(* Schneider Machine Expert - Basic project Proiect_final, file version 2.6.0.0 *)
(* ProjectInformations: Name=New project *)

HARDWARE
  Cpu 0: TM221CE16R
  ModuleExtensionObject 0: TM3AM6/G
  EthernetConfiguration: NetworkName=M221, IpAllocationMode=FixedAddress, IpAddress=0.0.0.0, SubnetMask=0.0.0.0
  SerialLineConfiguration: Baud=Baud19200, Parity=ParityEven, DataBits=DataBits8, StopBits=StopBits1, PhysicalMedium=PhysicalMediumRs485, TransmissionMode=TransmissionModeModbusRtu, SlaveId=1, Addressing=SlaveAddressing
  MastTask: UsePeriodScanMode=false, PeriodScan=100
  FastTask: Period=255
  CpuBehavior: StartingMode=StartAsPreviousState, AutoSaveRamOnEeprom=true, WatchdogPeriod=250

SYMBOLS  (address, symbol, comment, settings)
  %M0         "Plata_card"
  %M1         "Plata_cash"
  %M2         "Oltenia"
  %M3         "Moldova"
  %M4         "Transilvania"
  %M5         "Dobrogea"
  %M6         "Trece_banconte_de_50"
  %M7         "Trece_bancnote_de_5"
  %M8         "Trece_bancnote_de_10"
  %M9         "Trece_bancnote_de_1"
  %M10        "Plata_a_fost_facuta"
  %M11        "PLATA_CARD_A_FOST_FACUTA"
  %M12        "A_FOST_SELECTAT_CEVA"
  %C0         "Numarator_50_lei"
  %C1         "Numarator_10_lei"
  %C2         "Numarator_5_lei"
  %C3         "Numarator_1_leu"
  %I0.0       "Pornire selectie"
  %I0.1       "Plata_card"
  %I0.2       "Plata_cash"
  %I0.3       "Selecteaza_Oltenia"
  %I0.4       "Selecteaza_Moldova"
  %I0.5       "Selecteaza_Transilvania"
  %I0.6       "Selecteaza_Dobrogea"
  %I0.8       "SENZOR_A_FOST_LIVRAT_TICHETUL"
  %Q0.0       "S-a eliberat tichetul"
  %IW1.0      [Type=Type_4_20mA, Scope=Scope_Customized, Minimum=4000, Maximum=20000]
  %IW1.1      [Type=Type_4_20mA, Scope=Scope_Customized, Minimum=4000, Maximum=20000]

POU New POU
  (* SectionNumber=1 *)

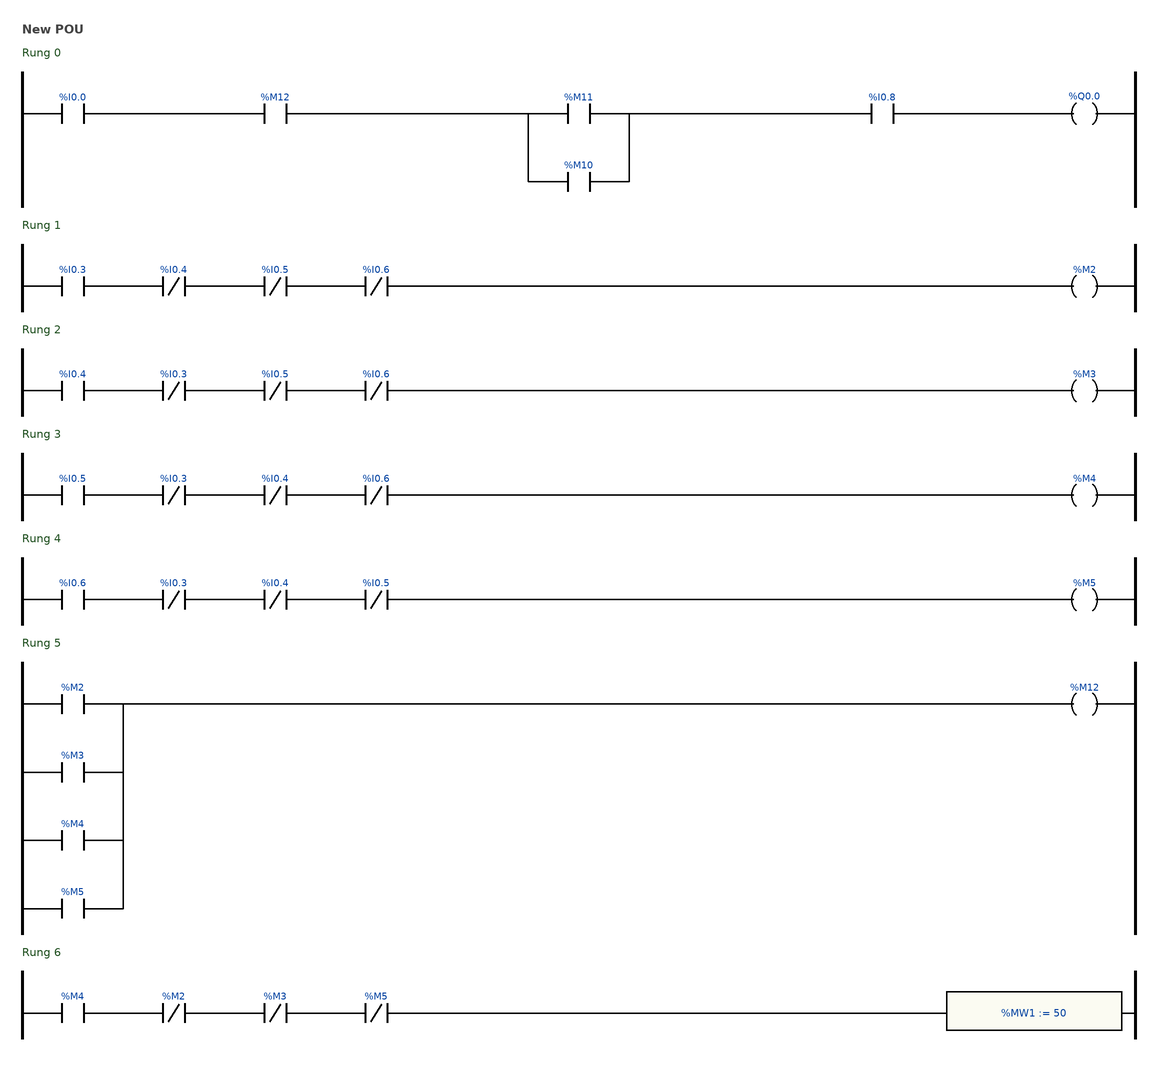

// Rung 0
  LD %I0.0
  AND %M12
  AND( %M11
  OR %M10
  )
  AND %I0.8
  ST %Q0.0
  // as ST:
  //   %Q0.0 := %I0.0 AND %M12 AND (%M11 OR %M10) AND %I0.8;

// Rung 1
  LD %I0.3
  ANDN %I0.4
  ANDN %I0.5
  ANDN %I0.6
  ST %M2
  // as ST:
  //   %M2 := %I0.3 AND NOT %I0.4 AND NOT %I0.5 AND NOT %I0.6;

// Rung 2
  LD %I0.4
  ANDN %I0.3
  ANDN %I0.5
  ANDN %I0.6
  ST %M3
  // as ST:
  //   %M3 := %I0.4 AND NOT %I0.3 AND NOT %I0.5 AND NOT %I0.6;

// Rung 3
  LD %I0.5
  ANDN %I0.3
  ANDN %I0.4
  ANDN %I0.6
  ST %M4
  // as ST:
  //   %M4 := %I0.5 AND NOT %I0.3 AND NOT %I0.4 AND NOT %I0.6;

// Rung 4
  LD %I0.6
  ANDN %I0.3
  ANDN %I0.4
  ANDN %I0.5
  ST %M5
  // as ST:
  //   %M5 := %I0.6 AND NOT %I0.3 AND NOT %I0.4 AND NOT %I0.5;

// Rung 5
  LD %M2
  OR %M3
  OR %M4
  OR %M5
  ST %M12
  // as ST:
  //   %M12 := %M2 OR %M3 OR %M4 OR %M5;

// Rung 6
  LD %M4
  ANDN %M2
  ANDN %M3
  ANDN %M5
  [ %MW1 := 50 ]
  // as ST:
  //   IF %M4 AND NOT %M2 AND NOT %M3 AND NOT %M5 THEN %MW1 := 50; END_IF;

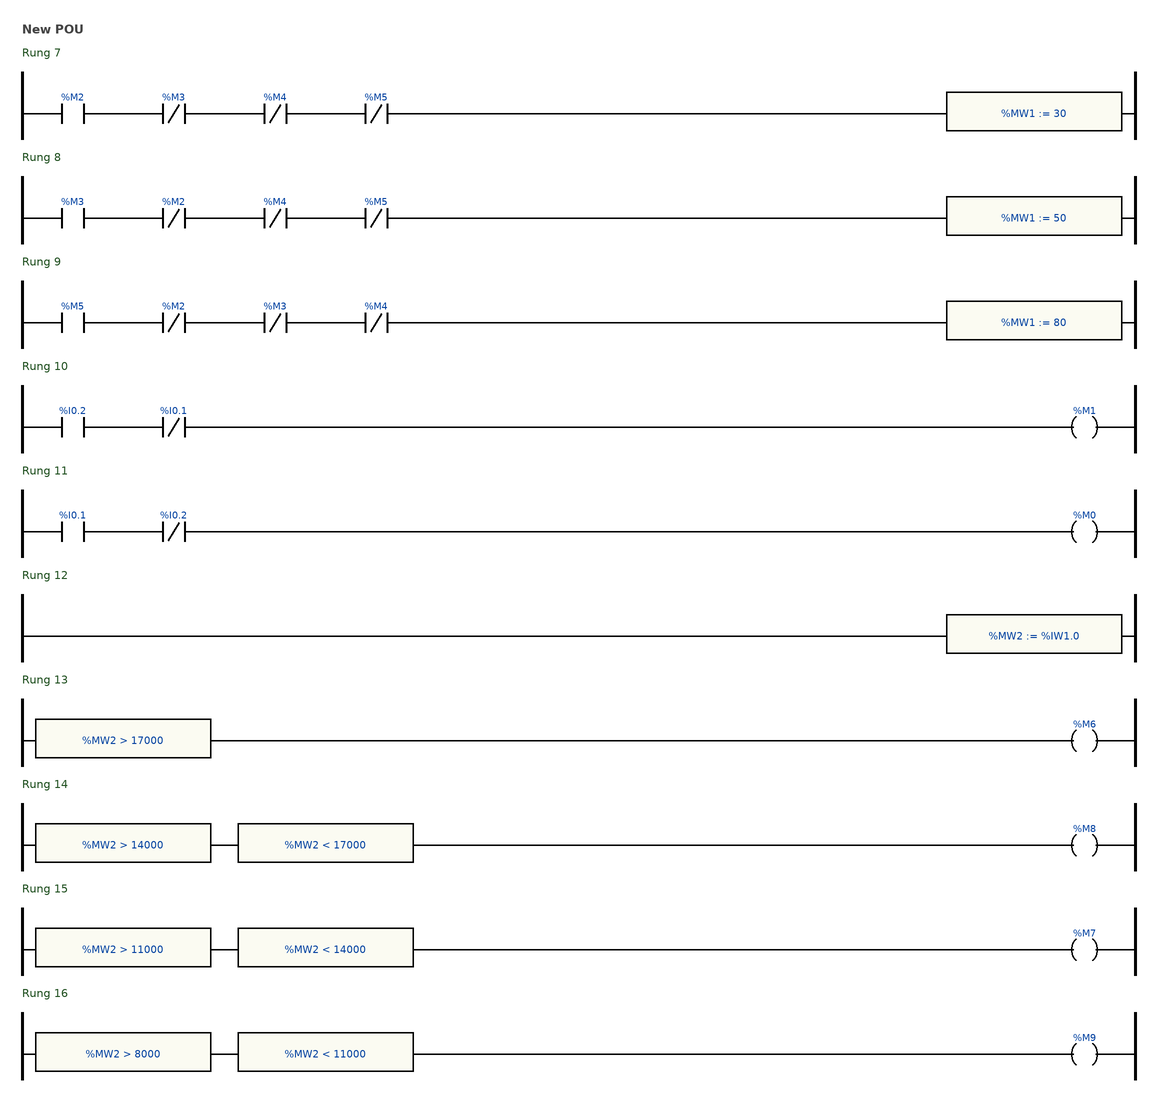

// Rung 7
  LD %M2
  ANDN %M3
  ANDN %M4
  ANDN %M5
  [ %MW1 := 30 ]
  // as ST:
  //   IF %M2 AND NOT %M3 AND NOT %M4 AND NOT %M5 THEN %MW1 := 30; END_IF;

// Rung 8
  LD %M3
  ANDN %M2
  ANDN %M4
  ANDN %M5
  [ %MW1 := 50 ]
  // as ST:
  //   IF %M3 AND NOT %M2 AND NOT %M4 AND NOT %M5 THEN %MW1 := 50; END_IF;

// Rung 9
  LD %M5
  ANDN %M2
  ANDN %M3
  ANDN %M4
  [ %MW1 := 80 ]
  // as ST:
  //   IF %M5 AND NOT %M2 AND NOT %M3 AND NOT %M4 THEN %MW1 := 80; END_IF;

// Rung 10
  LD %I0.2
  ANDN %I0.1
  ST %M1
  // as ST:
  //   %M1 := %I0.2 AND NOT %I0.1;

// Rung 11
  LD %I0.1
  ANDN %I0.2
  ST %M0
  // as ST:
  //   %M0 := %I0.1 AND NOT %I0.2;

// Rung 12
  LD 1
  [ %MW2 := %IW1.0 ]
  // as ST:
  //   %MW2 := %IW1.0;

// Rung 13
  LD [ %MW2 > 17000 ]
  ST %M6
  // as ST:
  //   %M6 := %MW2 > 17000;

// Rung 14
  LD [ %MW2 > 14000 ]
  AND [ %MW2 < 17000 ]
  ST %M8
  // as ST:
  //   %M8 := %MW2 > 14000 AND %MW2 < 17000;

// Rung 15
  LD [ %MW2 > 11000 ]
  AND [ %MW2 < 14000 ]
  ST %M7
  // as ST:
  //   %M7 := %MW2 > 11000 AND %MW2 < 14000;

// Rung 16
  LD [ %MW2 > 8000 ]
  AND [ %MW2 < 11000 ]
  ST %M9
  // as ST:
  //   %M9 := %MW2 > 8000 AND %MW2 < 11000;

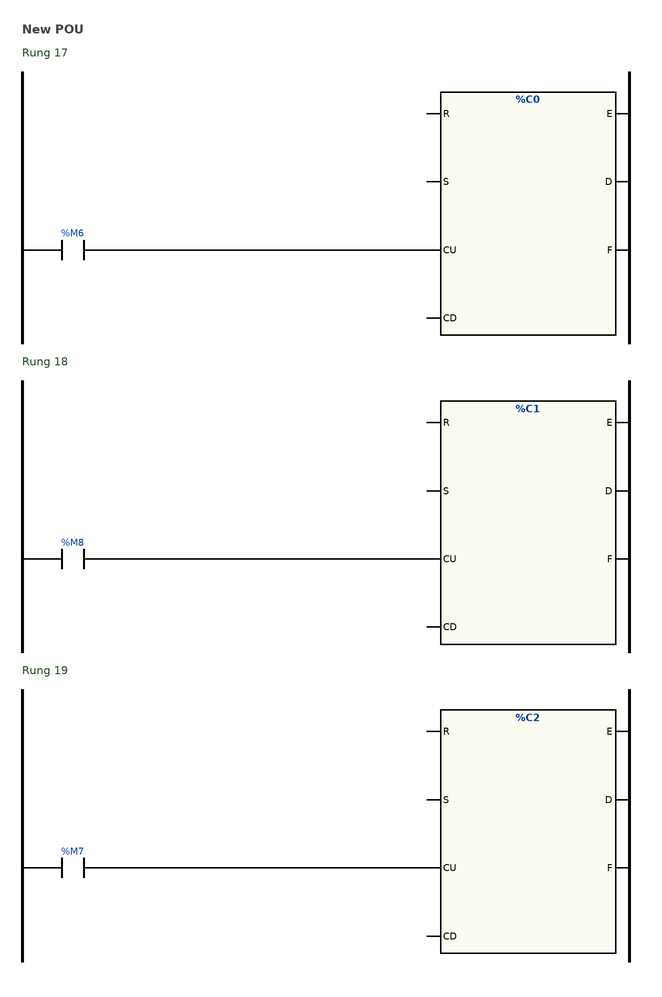

// Rung 17
  BLK %C0
  LD %M6
  CU
  END_BLK
  // as ST:
  //   %C0(CU := %M6);

// Rung 18
  BLK %C1
  LD %M8
  CU
  END_BLK
  // as ST:
  //   %C1(CU := %M8);

// Rung 19
  BLK %C2
  LD %M7
  CU
  END_BLK
  // as ST:
  //   %C2(CU := %M7);

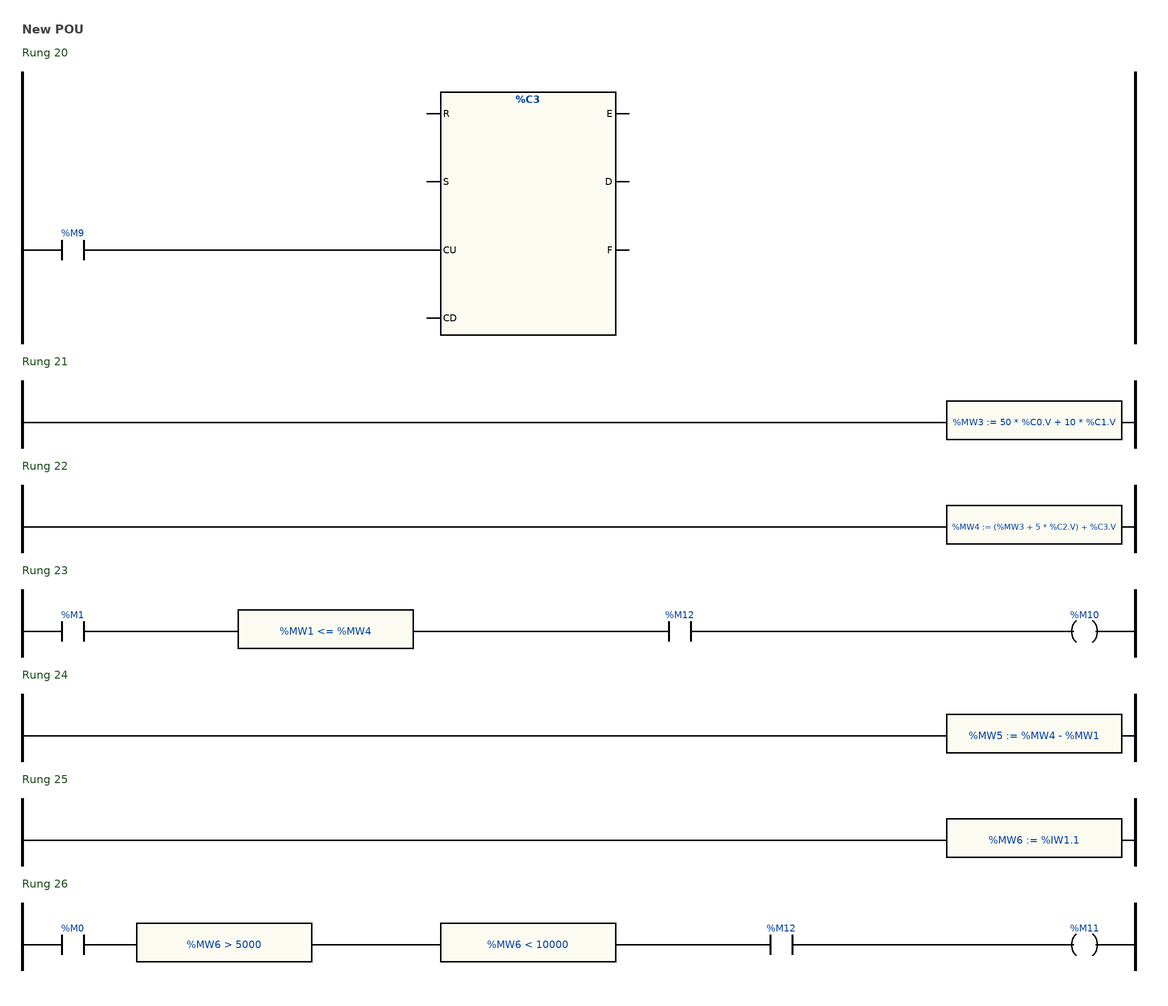

// Rung 20
  BLK %C3
  LD %M9
  CU
  END_BLK
  // as ST:
  //   %C3(CU := %M9);

// Rung 21
  LD 1
  [%MW3 := 50 * %C0.V + 10 * %C1.V]
  // as ST:
  //   %MW3 := 50 * %C0.V + 10 * %C1.V;

// Rung 22
  LD 1
  [%MW4 := (%MW3 + 5 * %C2.V) + %C3.V]
  // as ST:
  //   %MW4 := (%MW3 + 5 * %C2.V) + %C3.V;

// Rung 23
  LD %M1
  AND [ %MW1 <= %MW4 ]
  AND %M12
  ST %M10
  // as ST:
  //   %M10 := %M1 AND %MW1 <= %MW4 AND %M12;

// Rung 24
  LD 1
  [ %MW5 := %MW4 - %MW1 ]
  // as ST:
  //   %MW5 := %MW4 - %MW1;

// Rung 25
  LD 1
  [ %MW6 := %IW1.1 ]
  // as ST:
  //   %MW6 := %IW1.1;

// Rung 26
  LD %M0
  AND [ %MW6 > 5000 ]
  AND [ %MW6 < 10000 ]
  AND %M12
  ST %M11
  // as ST:
  //   %M11 := %M0 AND %MW6 > 5000 AND %MW6 < 10000 AND %M12;
